{attribute 'qualified_only'}
{attribute 'strict'}
TYPE E_FSM_Step :
(
	(* special steps *)
	NoStep := -32767,		// nessuno step
	Unknown := -32000,		// step sconosciuto
	
	(* Error steps *)
	NeOrError := -990,		// non abilitata o in errore
	Recovering := -980,		// azzeramento errori

	(* Stop *)
	Stop := 0,				// stop
	
	(* Cycle *)
	Running := 100,			// funzionamento nominale delle zone
		
	(* Stopping *)
	Stopping := 900			// fase di arresto
);
END_TYPE
//  NoStep = '-32767'
//  Unknown = '-32000'
//  NeOrError = '-990'
//  Recovering = '-980'

(* stored: Version 1.1.0.1
   EnumerationTextList E_FSM_Step: Id {64910d9b-75b9-0b71-293d-13ff2961142d} *)
